FUNCTION_BLOCK FB_Dictionary EXTENDS TNamedBase
VAR
	Keys : FB_StringList;
	Values : FB_TargList;
END_VAR

// Add item to list. TRUE if successful. 
METHOD PUBLIC AddItem : BOOL
VAR_INPUT
	Key : T_MaxString; // item key to add.
	Value : T_Arg;
END_VAR
IF Keys.Count <> Values.Count THEN
	LogWarning('Missmatch keys and values count. Clearing dictionary.');
	THIS^.Clear();
	RETURN;
END_IF
IF Keys.Count = GVL_List.LIST_SIZE THEN
	F_LogWarning(
		CONCAT(InstanceName, 'Dictionary is full.')
	);
	RETURN;
END_IF
IF Key = '' THEN
	LogWarning('key is null.');
	RETURN;
END_IF
IF Contains( Key )  THEN
	LogWarning('Key already exists in dictionary.');
	RETURN;
END_IF

IF Value.cbLen <= 0 THEN
	LogWarning('Value has no length.');
	RETURN;
END_IF

// Add the key.
IF NOT Keys.AddItem( Key ) THEN
	F_LogWarning(
		CONCAT(InstanceName, ' error adding key.')
	);
	RETURN;
END_IF
// add the value.
IF NOT Values.AddItem( Value ) THEN // if this fails, remove the key.
	LogWarning('Error adding value.');
	Keys.RemoveIndex( 
		INT_TO_UDINT( Keys.FindIndex( Key ) )
	);
	RETURN;
END_IF

AddItem := TRUE;
END_METHOD

// Removes all list items
METHOD PUBLIC Clear
Keys.Clear();
Values.Clear();
END_METHOD

// TRUE if Item is in FB_List.
METHOD PUBLIC Contains : BOOL
VAR_INPUT
	Key : T_MaxString; // Item to check.
END_VAR
VAR
	i : UINT := 0;
END_VAR
Contains := Keys.Contains ( Key );
END_METHOD

{attribute 'monitoring' := 'call'}
// Number of items in list.
PROPERTY PUBLIC Count : UDINT
GET
Count := Keys.Count;
END_GET
END_PROPERTY

// Return item in dictionary base on key.
METHOD PUBLIC Get : T_Arg
VAR_INPUT
	Key : T_MaxString;
END_VAR
THIS^.TryGet(Key, Get);
END_METHOD

PROPERTY PUBLIC ReferenceToThis : REFERENCE TO FB_Dictionary
GET
ReferenceToThis REF= THIS^;
END_GET
END_PROPERTY

//Remove the specified index. Shuffle remaining so list is intact.
METHOD PUBLIC Remove : BOOL
VAR_INPUT
	Key : T_MaxString;
END_VAR
IF Keys.Contains( Key ) THEN // invalid index request.
	LogWarning('Cannot remove key as not in dictionary.');
	RETURN;
END_IF

Values.RemoveIndex(
	INT_TO_UDINT( Keys.FindIndex( Key ) ) 
);

Keys.RemoveIndex( 
	INT_TO_UDINT( Keys.FindIndex( Key ) ) 
);

Remove := TRUE;
END_METHOD

// TRUE if successful and list item in sItem
METHOD PUBLIC TryGet : BOOL
VAR_IN_OUT CONSTANT
	Key : T_MaxString;
END_VAR
VAR_IN_OUT
	Value : T_Arg;
END_VAR
IF Keys.Contains( Key ) THEN
	Value := Values.GetIndex( 
				INT_TO_UDINT( Keys.FindIndex( Key ) ) 
			);
	TryGet := TRUE;
END_IF
END_METHOD

// TRUE if successful and list item in sItem
METHOD PUBLIC TryGetIndex : BOOL
VAR_INPUT
	Index : UDINT;
END_VAR
VAR_IN_OUT
	Key : T_MaxString;
	Value : T_Arg;
END_VAR
IF Index < Keys.Count THEN
	Key := Keys.GetIndex( Index );
	Value := Values.GetIndex( Index );
	TryGetIndex := TRUE;
END_IF
END_METHOD

// TRUE if successful. Returns value associated with first key that provides partial match
METHOD PUBLIC TryGetPartialKey : BOOL
VAR_IN_OUT CONSTANT
	PartialKey : T_MaxString;
END_VAR
VAR_IN_OUT
	Value : T_Arg;
END_VAR
IF Keys.ContainsPartial( PartialKey ) THEN
	Value := Values.GetIndex( 
				INT_TO_UDINT( Keys.FindIndexPartialKey( PartialKey ) ) 
			);
	TryGetPartialKey := TRUE;
END_IF
END_METHOD

END_FUNCTION_BLOCK

(* stored: Version 1.1.0.1, ProductVersion 3.1.4022.3
   POU FB_Dictionary: Id {c29a5ccc-af91-48ad-9b38-0f1964c51b1a}, SpecialFunc None
   Method AddItem: Id {7f6a3f31-76ca-43fd-91b7-7728f56d08a8}
   Method Clear: Id {6171b5ae-1e5a-4da3-8aae-f3f9b14b50f0}
   Method Contains: Id {d4b61f9c-9d80-41dc-973a-fcda4ce30650}
   Property Count: Id {44f257b5-c4fa-4cd1-8dc1-bdecfe5fa265}
   Get Get: Id {58e1d400-3be9-4148-b0a0-4123ff0c7bde}
   Method Get: Id {70d9cd8c-ffd0-4f6d-a5d4-d94f7bdee34a}
   Property ReferenceToThis: Id {fe01e567-8b69-499d-bb15-e6243979bb05}
   Get Get: Id {4723c871-a6a0-4092-af51-2c3e6a7a17b1}
   Method Remove: Id {6fb60066-ca81-4592-b347-e83cce4a9db9}
   Method TryGet: Id {57309371-ecb9-4896-9524-830ae1c28ddc}
   Method TryGetIndex: Id {ec616992-8a13-444b-bbce-5f2335c63e5a}
   Method TryGetPartialKey: Id {7941785e-7afc-4792-98ed-824c55eed538} *)
